(* PLC project Sin nombre, Desconocido Sin nombre 1 *)
(* stored: creationDateTime 2025-10-24T12:26:17, modificationDateTime 2025-10-25T13:14:10 *)

PROGRAM Lab2_OpenPLC
  VAR
    Btn_Control AT %IX0.0 : BOOL := FALSE;  (* Botón para iniciar/detener el aumento de presión. *)
    Presion AT %MW0.0 : INT := 300;  (* Variable de presión de la planta. *)
    LED_Emergencia AT %QX0.0 : BOOL := FALSE;  (* Control del LED (encendido = emergencia). *)
    Flag_Aumentar AT %QX0.1 : BOOL := FALSE;  (* Bandera de estado: aumento activo. *)
    Flag_Disminuir AT %QX0.2 : BOOL := FALSE;  (* Bandera de estado: disminución activa. *)
    Emergencia_Activa AT %QX0.3 : BOOL := FALSE;  (* Bandera que indica que el sistema está en modo de emergencia. *)
    Flag_Reloj_ON AT %QX0.4 : BOOL := FALSE;  (* Bandera de estado que mantiene el TON activo. *)
  END_VAR
  VAR
    Pulso : BOOL;  (* Señal de reloj (Base de tiempo para la tasa de 1 unidad/s) *)
    Aux_Trig : R_TRIG;  (* Bloque auxiliar para detectar flanco ascendente en Btn_Control *)
    SR_Aumentar : SR;  (* Establece el valor de Flag_Aumentar *)
    SR_Emergencia : SR;  (* Establece el valor de Emergencia_Activa *)
    SR_Disminuir : SR;  (* Establece el valor de Flag_Disminuir *)
    TON_Reloj : TON;  (* Permite generar el valor de Pulso *)
    R_TRIG_Reloj : R_TRIG;  (* Permite generar el valor de Pulso *)
    SR_Reloj : SR;  (* Permite generar el valor de Pulso *)
  END_VAR

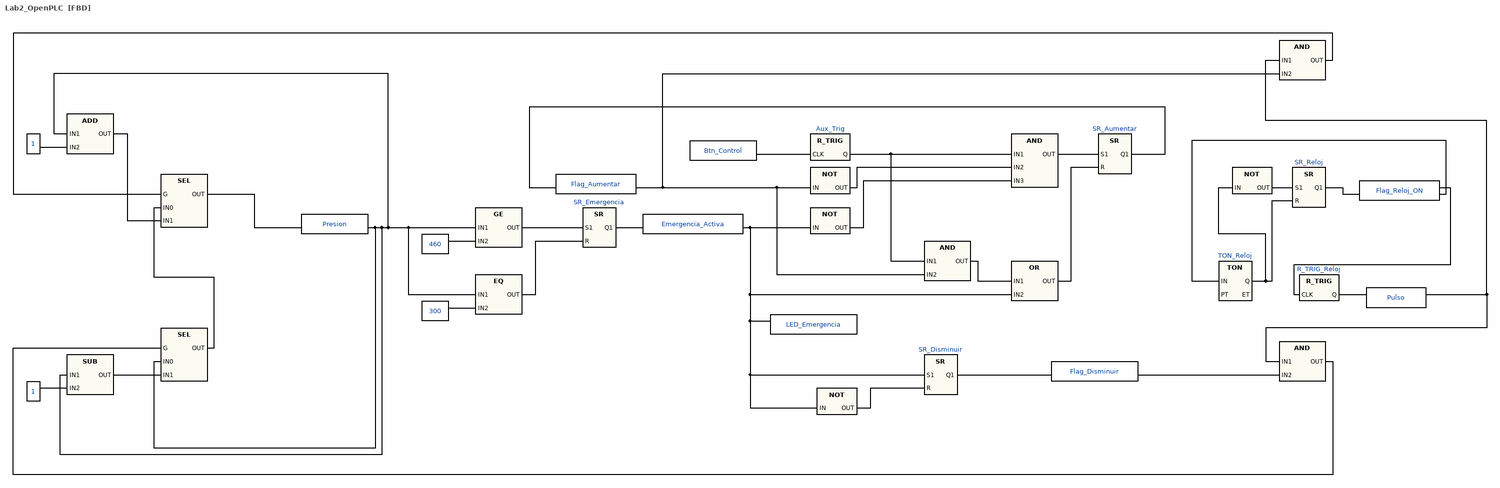
(* FBD diagram, written out as Structured Text *)
Aux_Trig(CLK := Btn_Control);
SR_Aumentar(S1 := Aux_Trig.Q AND NOT Flag_Aumentar AND NOT Emergencia_Activa, R := Aux_Trig.Q AND Flag_Aumentar OR Emergencia_Activa);
Flag_Aumentar := SR_Aumentar.Q1;
Presion := SEL(Pulso AND Flag_Aumentar, SEL(Pulso AND Flag_Disminuir, Presion, Presion - 1), Presion + 1);
SR_Emergencia(S1 := Presion >= 460, R := Presion = 300);
Emergencia_Activa := SR_Emergencia.Q1;
LED_Emergencia := Emergencia_Activa;
SR_Disminuir(S1 := Emergencia_Activa, R := NOT Emergencia_Activa);
Flag_Disminuir := SR_Disminuir.Q1;
TON_Reloj(IN := Flag_Reloj_ON);
SR_Reloj(S1 := NOT TON_Reloj.Q, R := TON_Reloj.Q);
Flag_Reloj_ON := SR_Reloj.Q1;
R_TRIG_Reloj(CLK := Flag_Reloj_ON);
Pulso := R_TRIG_Reloj.Q;
END_PROGRAM

CONFIGURATION Config0
  RESOURCE Res0 ON PLC
    TASK task0(INTERVAL := T#20ms, PRIORITY := 0);
    PROGRAM instance0 WITH task0 : Lab2_OpenPLC;
  END_RESOURCE
END_CONFIGURATION
